RoboDK station: movimiento_mocap.rdk

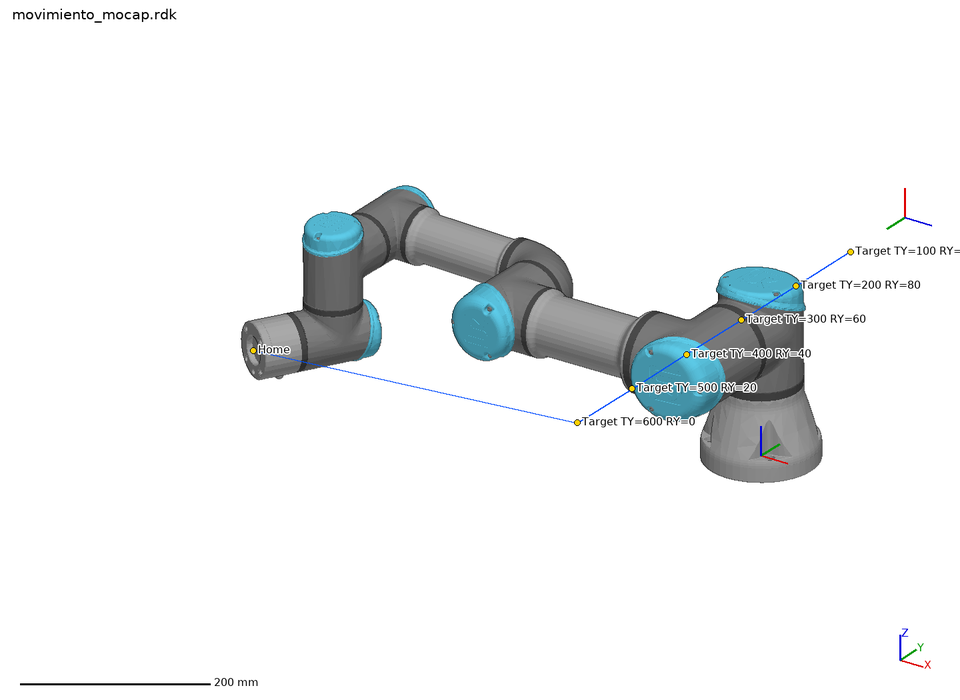
[picture v0: the station drawn from its stored meshes, robots at their saved joint values, targets as dots, program paths as lines]
Station movimiento_mocap (saved by RoboDK 5.5.2). Poses are relative to the parent item; angles as X-Y-Z fixed-axis rotations.
  - frame UR3e Base at (0, 0, 0) mm
    - robot UR3e: 6 axes, payload 3 kg, reach 500 mm, repeatability 0.03 mm, weight 11 kg
        modified DH rows (alpha deg, a mm, theta deg, d mm): 0, 0, 0, 151.9; 90, 0, 180, 0; 0, 243.55, 0, 0; 0, 213.2, 0, 131.05; -90, 0, 0, 85.35; 90, 0, 180, 92.1
        joint limits [-360, -360, -360, -360, -360, -360] to [360, 360, 360, 360, 360, 360]; home [0, -90, -90, 0, 90, 0]; saved at [0, 0.865, -1.845, 0.94, 30, 0.034]
    - frame B0 frame at (150, 50, 300) mm, rotated rx 0 ry -90 rz 180 deg
      - target Home (joint target) at (-233.45, 260.81, -652.8) mm, rotated rx -173.72 ry -60 rz 90 deg; joints [0, 0.865, -1.845, 0.94, 30, 0.034] of UR3e
      - target Target TY=600 RY=0 (Cartesian target) at (0, 600, 0) mm; joints [-147.982, -180, 0, -180, -117.982, 0] of UR3e
      - target Target TY=500 RY=20 (Cartesian target) at (0, 500, 0) mm, rotated rx 0 ry 20 rz 0 deg; joints [-147.982, -180, 0, -180, -117.982, 0] of UR3e
      - target Target TY=400 RY=40 (Cartesian target) at (0, 400, 0) mm, rotated rx 0 ry 40 rz 0 deg; joints [-147.982, -180, 0, -180, -117.982, 0] of UR3e
      - target Target TY=300 RY=60 (Cartesian target) at (0, 300, 0) mm, rotated rx 0 ry 60 rz 0 deg; joints [-147.982, -180, 0, -180, -117.982, 0] of UR3e
      - target Target TY=200 RY=80 (Cartesian target) at (0, 200, 0) mm, rotated rx 0 ry 80 rz 0 deg; joints [-147.982, -180, 0, -180, -117.982, 0] of UR3e
      - target Target TY=100 RY=100 (Cartesian target) at (0, 100, 0) mm, rotated rx 180 ry 80 rz 180 deg; joints [-147.982, -180, 0, -180, -117.982, 0] of UR3e
  - program My Prog (7 instructions, listed below)
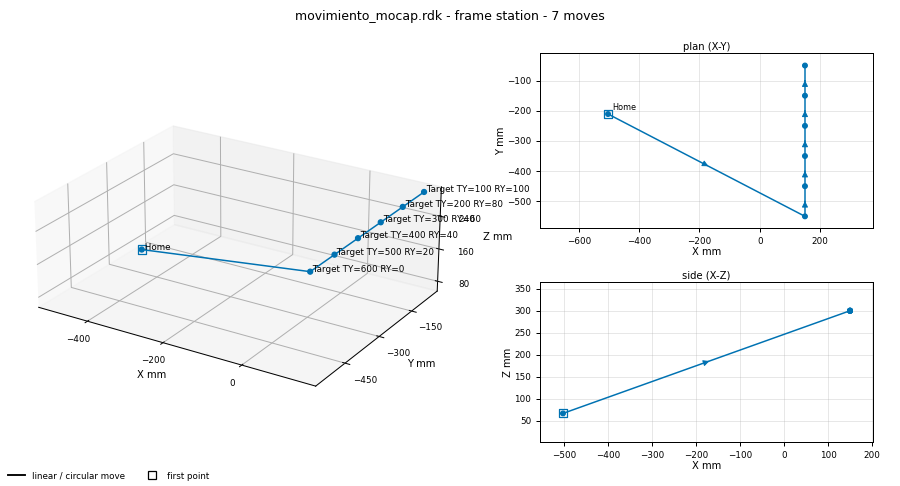
[picture p0: tool path of movimiento_mocap.rdk in frame station, 7 of 7 moves have a stored position in this frame; points joined in program order, loops and branches not executed]

--- program My Prog (robot UR3e) ---
  MoveJ (Home)
  MoveL (Target TY=600 RY=0)
  MoveL (Target TY=500 RY=20)
  MoveL (Target TY=400 RY=40)
  MoveL (Target TY=300 RY=60)
  MoveL (Target TY=200 RY=80)
  MoveL (Target TY=100 RY=100)
